# EPICS autosave request: soft_iocs/galil_DMC/iocBoot/iocgalil_DMC_E02/GalilTest_18ID_DMC_E02Positions.req
$(P)9.DVAL
$(P)10.DVAL
$(P)11.DVAL
$(P)12.DVAL
$(P)13.DVAL
$(P)14.DVAL
$(P)15.DVAL
$(P)16.DVAL
